TYPE ST_PistonRange :
STRUCT
	fPistonPosMin : LREAL :=0;
	fPistonPosMax : LREAL :=0.5;
END_STRUCT
END_TYPE

(* stored: Version 1.1.0.1, ProductVersion 3.1.4024.10
   DUT ST_PistonRange: Id {917d97e8-5c6e-415f-bdae-656681d21934} *)
